# EPICS autosave request: softGlueApp/Db/histScalerDma_settings.req
$(P)$(Q)histScalerDmaEnable
$(P)$(Q)histScalerDma.SCAN
